FUNCTION F_HE_SATT_IsUsableFilter : BOOL
VAR_INPUT
    iFilter : I_HE_SATT_Filter;
END_VAR

END_FUNCTION

(* stored: Version 1.1.0.1
   POU F_HE_SATT_IsUsableFilter: Id {71ef2912-7b5e-4b3f-91f1-0c5f670d46d4}, SpecialFunc None *)
